{attribute addProperty BoxType "EL1259-0000-0017"}
{attribute addProperty Id "MTO_Inputs_ChannelAT %I*ARRAY[0..7] OF MTO_Inputs_Channel_5AD475AF8721090MTI_Inputs_10x_ChannelAT %I*ARRAY[0..84] OF MTI_Inputs_10x_Channel_D2104A6045285660MTO_Outputs_10x_ChannelAT %Q*ARRAY[0..84] OF MTO_Outputs_10x_Channel_24D255B145285660MTI_Outputs_ChannelAT %Q*ARRAY[0..7] OF MTI_Outputs_Channel_DD76C79810961370WcStateAT %I*WcState_98A4DF7520.250InfoDataAT %I*InfoData_0BDED7BF144180"}
{attribute addProperty CRC "1774539063"}
{attribute addProperty SizeInBites "11170"}
{attribute addProperty SizeInBytes "1396.25"}
TYPE EL1259_E12F1426 :
STRUCT
	{attribute addProperty Name "MTO_Inputs_Channel"}
	MTO_Inputs_Channel : ARRAY[0..7] OF MTO_Inputs_Channel_5AD475AF;
	{attribute addProperty Name "MTI_Inputs_10x_Channel"}
	MTI_Inputs_10x_Channel : ARRAY[0..84] OF MTI_Inputs_10x_Channel_D2104A60;
	{attribute addProperty Name "MTO_Outputs_10x_Channel"}
	MTO_Outputs_10x_Channel : ARRAY[0..84] OF MTO_Outputs_10x_Channel_24D255B1;
	{attribute addProperty Name "MTI_Outputs_Channel"}
	MTI_Outputs_Channel : ARRAY[0..7] OF MTI_Outputs_Channel_DD76C798;
	{attribute addProperty Name "WcState"}
	WcState : WcState_98A4DF75;
	{attribute addProperty Name "InfoData"}
	InfoData : InfoData_0BDED7BF;
END_STRUCT
END_TYPE

(* stored: Version 1.2.0.0, ProductVersion 3.1.4024.9
   DUT EL1259_E12F1426: Id {0a8ca180-34e2-421b-8b1b-ff818b7ee81c} *)
